(* Logix 5000 project; controller CTRL_PLC_V30 vendor 1 type 14 code 212 rev 34.11; software revision 34.02; part 2 of 2 *)
(* tags used below, declared in another part *)
   Aantal_RondjesT1 : DINT;
   Aantal_RondjesT2 : DINT;
   As_Test1_CTRL : AXIS_CIP_DRIVE;
   As_Test2_CTRL : AXIS_CIP_DRIVE;
   AsTest1Accel : REAL;
   AsTest1Snelheid : REAL;
   AsTest1StartPos : REAL;
   AsTest1StopPos : REAL;
   AsTest2Accel : REAL;
   AsTest2Snelheid : REAL;
   AsTest2StartPos : REAL;
   AsTest2StopPos : REAL;
   BOOL : BOOL;
   Drive_SAFE_OFF1 : ALIAS FOR DRIVER:SO.SafeTorqueOff1;
   Drive_SAFE_OFF2 : ALIAS FOR DRIVER:SO.SafeTorqueOff2;
   ERROR : BOOL;
   ERROR_1 : BOOL;
   ERROR_2 : BOOL;
   ESTP_ACTIVATED : BOOL;
   HomeT1 : ALIAS FOR IOP_HMI_BT[0].2;
   HomeT2 : ALIAS FOR IOP_HMI_BT[1].2;
   ILB_RESET_SAFETY1 : BOOL;
   ILG_CTRL_VOLT1 : BOOL;
   IO_SPLC_TO_CTRL : UDT_COMM_SPLC_TO_CTRL;
   IOP_HMI_BT : DINT[2];
   IOP_HMI_REAL : REAL[20];
   MDA_DATACHOICE : INT;
   MDB_DATACHOICE : INT;
   Motioncontrol13 : MOTION_INSTRUCTION;
   Motioncontrol14 : MOTION_INSTRUCTION;
   Motioncontrol21 : MOTION_INSTRUCTION;
   Motioncontrol26 : MOTION_INSTRUCTION;
   Motioncontrol27 : MOTION_INSTRUCTION;
   Motioncontrol3 : MOTION_INSTRUCTION;
   Motioncontrol30 : MOTION_INSTRUCTION;
   Motioncontrol4 : MOTION_INSTRUCTION;
   Motionctrl1 : MOTION_INSTRUCTION;
   Motionctrl2 : MOTION_INSTRUCTION;
   Motionstart1 : MOTION_INSTRUCTION;
   Motionstartl2 : MOTION_INSTRUCTION;
   OvertravelFault : BOOL;
   OvertravelFault2 : BOOL;
   QOP_HMI_BT : DINT[10];
   QOP_HMI_GRAPH1_HDR : REAL[10];
   QOP_HMI_GRAPH1_LINE1_DATAX : REAL[800];
   QOP_HMI_GRAPH1_LINE1_DATAY : REAL[800];
   QOP_HMI_GRAPH1_LINE1_HDR : REAL[10];
   QOP_HMI_GRAPH1_LINE2_DATAY : REAL[800];
   QOP_HMI_GRAPH2_HDR : REAL[10];
   QOP_HMI_GRAPH2_LINE1_DATAX : REAL[800];
   QOP_HMI_GRAPH2_LINE1_DATAY : REAL[800];
   QOP_HMI_GRAPH2_LINE2_DATAY : REAL[800];
   RondjesT1 : REAL;
   RondjesT2 : REAL;
   SAF_RESET_KNOP : BOOL;
   Safeovertravel1 : REAL;
   Safeovertravel2 : REAL;
   SAFETY_DOOR1_OPEN : BOOL;
   SAFETY_DOOR2_OPEN : BOOL;
   StartG : ALIAS FOR RIO_CTRL:3:I.0;
   StartLampje : ALIAS FOR RIO_CTRL:5:O.0;
   StartT1 : ALIAS FOR IOP_HMI_BT[0].0;
   StartT2 : ALIAS FOR IOP_HMI_BT[1].0;
   StateT1Routine : DINT;
   StateT2Routine : DINT;

   StopLampje : ALIAS FOR RIO_CTRL:5:O.1;
   StopR : ALIAS FOR RIO_CTRL:3:I.1;
   StopT1 : ALIAS FOR IOP_HMI_BT[0].1;
   StopT2 : ALIAS FOR IOP_HMI_BT[1].1;
   TEST_1x : BOOL;
   TIME_LATCH : BOOL; {access Read Only}
   Timer1 : TIMER := (PRE := 2);
   TIMER10 : TIMER := (PRE := 10000); {access Read Only}
   Timer2 : TIMER := (PRE := 2);
   Timeras1 : FBD_TIMER := (TimerEnable := 1, PRE := 9000, Reset := 1, ACC := 7821, EN := 1, TT := 1);
   Timeras2 : FBD_TIMER;
   Timeras3 : FBD_TIMER;
   Timeras4 : FBD_TIMER;
   Timeras5 : FBD_TIMER;
   Timeras6 : FBD_TIMER := (TimerEnable := 1, PRE := 200, Reset := 1, ACC := 151, EN := 1, TT := 1);
   Timeras7 : FBD_TIMER := (TimerEnable := 1, PRE := 9000, Reset := 1, ACC := 5957, EN := 1, TT := 1);
   Timeras8 : FBD_TIMER := (TimerEnable := 1, PRE := 9000, Reset := 1, ACC := 5010, EN := 1, TT := 1);
   Timeras9 : FBD_TIMER := (TimerEnable := 1, PRE := 9000, Reset := 1, ACC := 5001, EN := 1, TT := 1);
END_VAR

PROGRAM DataVersturen   (* main routine DataPLC *)
VAR
   FORLOOPINT : INT := 400; {access None}
   FORLOOPINT2 : DINT := 800; {access None}
   GRAPH1_LATESTX : INT; {access None}
   IDLE : DINT;
   POSITION1_INT : INT; {access None}
   POSITION2_INT : INT := 799; {access None}
   STEPSIZE2_LINE1 : REAL := -0.02; {access None}
   STEPSIZE_LINE1 : REAL := 11.875; {access None}
   TIMERMOV : TIMER := (PRE := 500, ACC := 10);
END_VAR

ROUTINE DataPLC   (* ladder *)
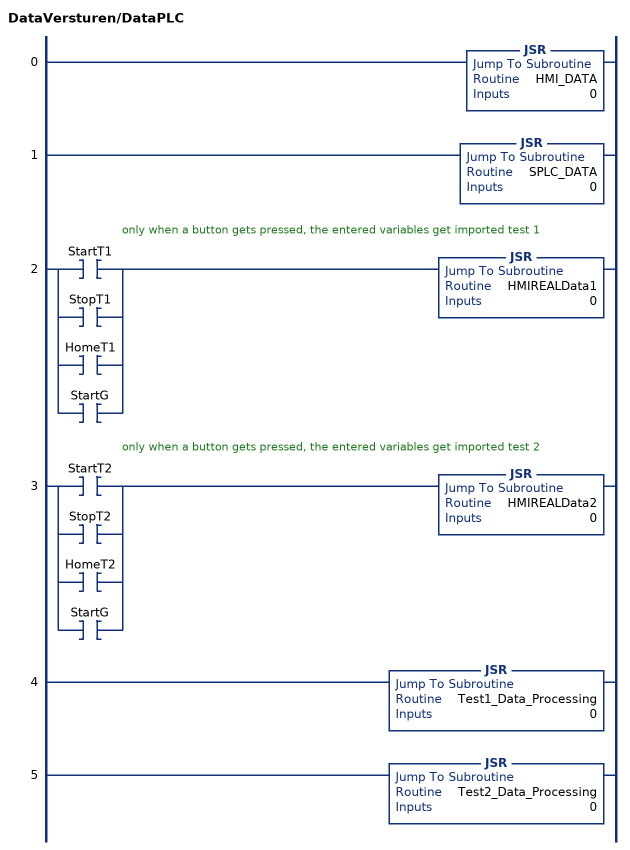
   0: JSR(HMI_DATA,0);
   1: JSR(SPLC_DATA,0);
   // only when a button gets pressed, the entered variables get imported test 1
   2: [XIC(StartT1) ,[XIC(StopT1) ,[XIC(HomeT1) ,XIC(StartG) ] ] ]JSR(HMIREALData1,0);
   // only when a button gets pressed, the entered variables get imported test 2
   3: [XIC(StartT2) ,[XIC(StopT2) ,[XIC(HomeT2) ,XIC(StartG) ] ] ]JSR(HMIREALData2,0);
   4: JSR(Test1_Data_Processing,0);
   5: JSR(Test2_Data_Processing,0);
END_ROUTINE

ROUTINE HMI_DATA   (* ladder *)
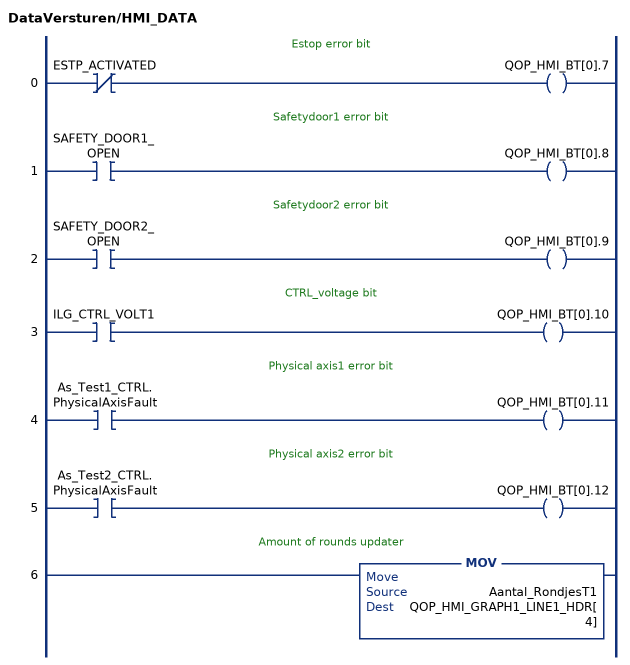
   // Estop error bit
   0: XIO(ESTP_ACTIVATED)OTE(QOP_HMI_BT[0].7);
   // Safetydoor1 error bit
   1: XIC(SAFETY_DOOR1_OPEN)OTE(QOP_HMI_BT[0].8);
   // Safetydoor2 error bit
   2: XIC(SAFETY_DOOR2_OPEN)OTE(QOP_HMI_BT[0].9);
   // CTRL_voltage bit
   3: XIC(ILG_CTRL_VOLT1)OTE(QOP_HMI_BT[0].10);
   // Physical axis1 error bit
   4: XIC(As_Test1_CTRL.PhysicalAxisFault)OTE(QOP_HMI_BT[0].11);
   // Physical axis2 error bit
   5: XIC(As_Test2_CTRL.PhysicalAxisFault)OTE(QOP_HMI_BT[0].12);
   // Amount of rounds updater
   6: MOV(Aantal_RondjesT1,QOP_HMI_GRAPH1_LINE1_HDR[4]);
END_ROUTINE

ROUTINE HMIREALData1   (* ladder *)
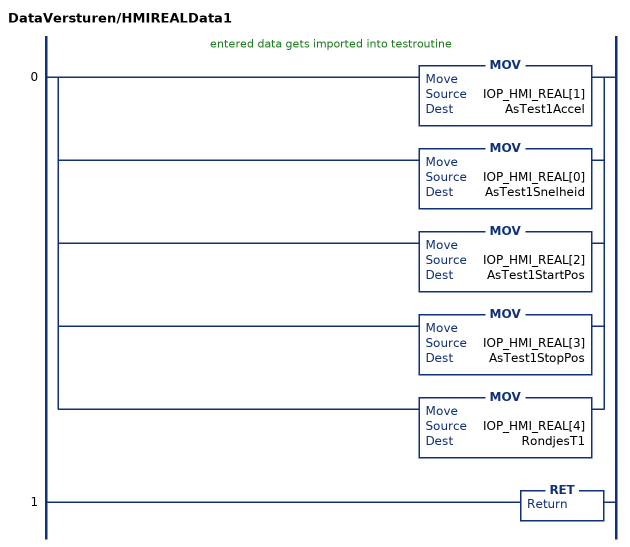
   // entered data gets imported into testroutine
   0: [MOV(IOP_HMI_REAL[1],AsTest1Accel) ,[MOV(IOP_HMI_REAL[0],AsTest1Snelheid) ,[MOV(IOP_HMI_REAL[2],AsTest1StartPos) ,[MOV(IOP_HMI_REAL[3],AsTest1StopPos) ,MOV(IOP_HMI_REAL[4],RondjesT1) ] ] ] ];
   1: RET();
END_ROUTINE

ROUTINE HMIREALData2   (* ladder *)
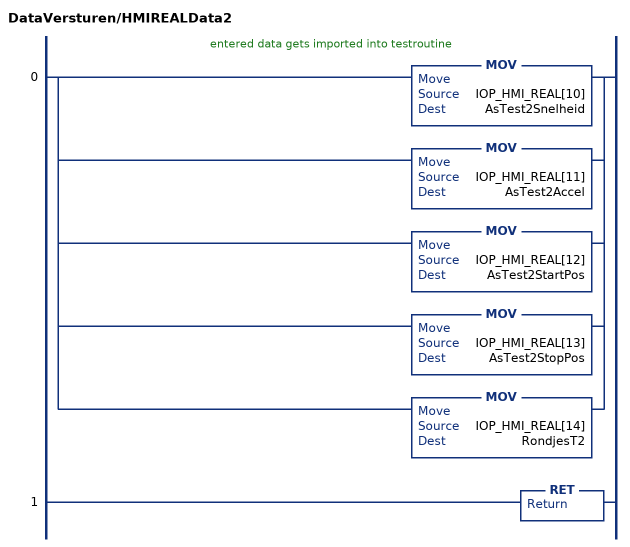
   // entered data gets imported into testroutine
   0: [MOV(IOP_HMI_REAL[10],AsTest2Snelheid) ,[MOV(IOP_HMI_REAL[11],AsTest2Accel) ,[MOV(IOP_HMI_REAL[12],AsTest2StartPos) ,[MOV(IOP_HMI_REAL[13],AsTest2StopPos) ,MOV(IOP_HMI_REAL[14],RondjesT2) ] ] ] ];
   1: RET();
END_ROUTINE

ROUTINE SPLC_DATA   (* ladder *)
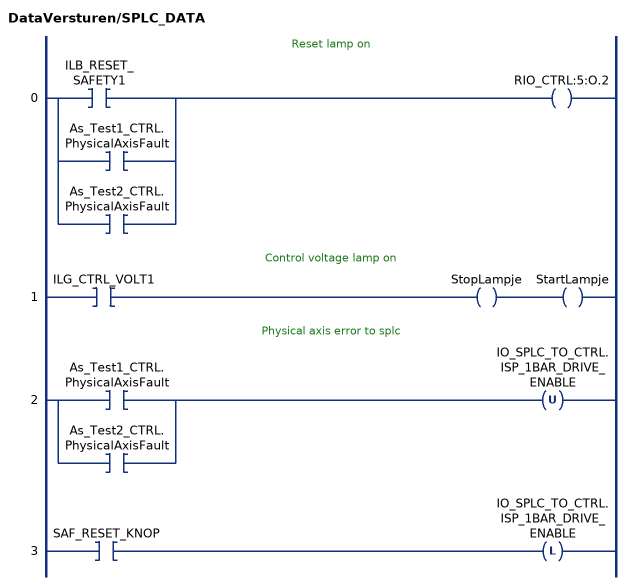
   // Reset lamp on
   0: [XIC(ILB_RESET_SAFETY1) ,[XIC(As_Test1_CTRL.PhysicalAxisFault) ,XIC(As_Test2_CTRL.PhysicalAxisFault) ] ]OTE(RIO_CTRL:5:O.2);
   // Control voltage lamp on
   1: XIC(ILG_CTRL_VOLT1)OTE(StopLampje)OTE(StartLampje);
   // Physical axis error to splc
   2: [XIC(As_Test1_CTRL.PhysicalAxisFault) ,XIC(As_Test2_CTRL.PhysicalAxisFault) ]OTU(IO_SPLC_TO_CTRL.ISP_1BAR_DRIVE_ENABLE);
   3: XIC(SAF_RESET_KNOP)OTL(IO_SPLC_TO_CTRL.ISP_1BAR_DRIVE_ENABLE);
END_ROUTINE

ROUTINE Test1_Data_Processing   (* structured text *)
   // wanneer state voltooid, dan naar volgende state
   
   CASE StateT1Routine OF
   	0: // idle state
   
   	1: // runs one time when subroutine starts
   	POSITION1_INT := 0;
   	FOR FORLOOPINT := 0 TO 799 BY 1 DO
   		QOP_HMI_GRAPH1_LINE1_DATAY[FORLOOPINT] := 0;		// emptying Array
   		QOP_HMI_GRAPH1_LINE2_DATAY[FORLOOPINT] := 0;		// emptying Array
   	END_FOR;
   	StateT1Routine := 2; // go to T1 state 2
   
   	2: // calculate steppsize
   	STEPSIZE_LINE1 := (AsTest1StopPos - AsTest1StartPos)/800;
   	STEPSIZE_LINE1 := STEPSIZE_LINE1 -0.0;
   	QOP_HMI_GRAPH1_LINE1_DATAX[0]:= AsTest1StartPos + 0.1;
   	FOR FORLOOPINT := 1 TO 799 BY 1 DO
   		QOP_HMI_GRAPH1_LINE1_DATAX[FORLOOPINT] := QOP_HMI_GRAPH1_LINE1_DATAX[FORLOOPINT-1]+STEPSIZE_LINE1;		// emtying Array
   	END_FOR;
   	QOP_HMI_GRAPH1_LINE1_DATAX[799]:= AsTest1StopPos - 0.1;
   	QOP_HMI_GRAPH1_HDR[2] := AsTest1StartPos;
   	QOP_HMI_GRAPH1_HDR[3]  :=AsTest1StopPos;
   	POSITION1_INT := 0;
   	StateT1Routine := 21;	// go to Test1Routine home sequence
   
   	6: // recording Data
   	StateT1Routine := 50 + MDA_DATACHOICE;
   
   	11:	// recording data
   	POSITION1_INT := 799;			//setting value ready for next state
   	StateT1Routine := 60 + MDA_DATACHOICE;
   
   	12: //changing graph setting
   	POSITION1_INT := 0;
   	QOP_HMI_GRAPH1_HDR[5] := 2;		// setting Ymax to a low value
   	FOR FORLOOPINT := 0 TO 399 BY 1 DO				// setting graph hight
   		IF QOP_HMI_GRAPH1_LINE1_DATAY[FORLOOPINT] > QOP_HMI_GRAPH1_HDR[5] THEN
   			QOP_HMI_GRAPH1_HDR[5] := QOP_HMI_GRAPH1_LINE1_DATAY[FORLOOPINT];
   		END_IF;
   	END_FOR;
   	FOR FORLOOPINT := 0 TO 399 BY 1 DO
   		IF QOP_HMI_GRAPH1_LINE2_DATAY[FORLOOPINT] > QOP_HMI_GRAPH1_HDR[5] THEN
   			QOP_HMI_GRAPH1_HDR[5] := QOP_HMI_GRAPH1_LINE2_DATAY[FORLOOPINT];
   		END_IF;
   	END_FOR;
   	IF (AsTest1StopPos - AsTest1StartPos)> 600 THEN // choosing graph x axis steppsize
   	QOP_HMI_GRAPH1_HDR[6]:= 20;
   	ELSIF (AsTest1StopPos - AsTest1StartPos)> 400 THEN
   	QOP_HMI_GRAPH1_HDR[6]:= 10;
   	ELSE
   	QOP_HMI_GRAPH1_HDR[6]:= 1;
   	END_IF;
   	IF QOP_HMI_GRAPH1_HDR[5] > 500 THEN				// choosing graph y axis steppsize
   	QOP_HMI_GRAPH1_HDR[7] := 50;
   	ELSIF QOP_HMI_GRAPH1_HDR[5] > 200 THEN
   	QOP_HMI_GRAPH1_HDR[7] := 25;
   	ELSIF QOP_HMI_GRAPH1_HDR[5] > 60 THEN
   	QOP_HMI_GRAPH1_HDR[7] := 5;
   	ELSE
   	QOP_HMI_GRAPH1_HDR[7] := 1;
   	END_IF;
   	StateT1Routine := 13; // go to Test1Routine state 13
   
   	14:	// check if all data has been sent to HMI
   	StateT1Routine := 15; // go to Test1Routine state 15
   
   	50:  // motion process
   	IF Motioncontrol3.PC THEN StateT1Routine := 10;	END_IF;
   
   	51: // Data of torque reference
   	IF As_Test1_CTRL.ActualPosition >= QOP_HMI_GRAPH1_LINE1_DATAX[POSITION1_INT] THEN
   		QOP_HMI_GRAPH1_LINE1_DATAY[POSITION1_INT]:= ABS(As_Test1_CTRL.TorqueReference);
   		POSITION1_INT := POSITION1_INT + 1;
   	END_IF;
   	IF POSITION1_INT > 799 OR Motioncontrol3.PC THEN
   		StateT1Routine := 10; // go to Test1Routine state 10
   	END_IF;
   
   	52: // Data of current reference
   	IF As_Test1_CTRL.ActualPosition >= QOP_HMI_GRAPH1_LINE1_DATAX[POSITION1_INT] THEN
   		QOP_HMI_GRAPH1_LINE1_DATAY[POSITION1_INT]:= ABS(As_Test1_CTRL.CurrentReference);
   		POSITION1_INT := POSITION1_INT + 1;
   
   	END_IF;
   	IF POSITION1_INT > 799 OR Motioncontrol3.PC THEN
   		StateT1Routine := 10; // go to Test1Routine state 10
   	END_IF;
   
   	53: // Data of actual velocity
   	IF As_Test1_CTRL.ActualPosition >= QOP_HMI_GRAPH1_LINE1_DATAX[POSITION1_INT] THEN
   		QOP_HMI_GRAPH1_LINE1_DATAY[POSITION1_INT]:= ABS(As_Test1_CTRL.ActualVelocity);
   		POSITION1_INT := POSITION1_INT + 1;
   
   	END_IF;
   	IF POSITION1_INT > 799 OR Motioncontrol3.PC THEN
   		StateT1Routine := 10; // go to Test1Routine state 10
   	END_IF;
   
   	60: // motion process
   	IF Motioncontrol4.PC THEN StateT1Routine := 12;	END_IF;
   
   	61: //TorqueReference
   	IF As_Test1_CTRL.ActualPosition <= QOP_HMI_GRAPH1_LINE1_DATAX[POSITION1_INT] THEN
   		QOP_HMI_GRAPH1_LINE2_DATAY[POSITION1_INT]:= ABS(As_Test1_CTRL.TorqueReference);
   		POSITION1_INT := POSITION1_INT - 1;
   	END_IF;
   	IF POSITION1_INT < 0 OR Motioncontrol4.PC THEN
   		StateT1Routine := 12; // go to T1 state 12
   	END_IF;
   
   	62: //CurrentReference
   	IF As_Test1_CTRL.ActualPosition <= QOP_HMI_GRAPH1_LINE1_DATAX[POSITION1_INT] THEN
   		QOP_HMI_GRAPH1_LINE2_DATAY[POSITION1_INT]:= ABS(As_Test1_CTRL.CurrentReference);
   		POSITION1_INT := POSITION1_INT - 1;
   	END_IF;
   	IF POSITION1_INT < 0 OR Motioncontrol4.PC THEN
   		StateT1Routine := 12; // go to T1 state 12
   	END_IF;
   
   	63: //ActualVelocity
   	IF As_Test1_CTRL.ActualPosition <= QOP_HMI_GRAPH1_LINE1_DATAX[POSITION1_INT] THEN
   		QOP_HMI_GRAPH1_LINE2_DATAY[POSITION1_INT]:= ABS(As_Test1_CTRL.ActualVelocity);
   		POSITION1_INT := POSITION1_INT - 1;
   	END_IF;
   	IF POSITION1_INT < 0 OR Motioncontrol4.PC THEN
   		StateT1Routine := 12; // go to T1 state 12
   	END_IF;
   
   END_CASE;
END_ROUTINE

ROUTINE Test2_Data_Processing   (* structured text *)
   // wanneer state voltooid, dan naar volgende state
   CASE StateT2Routine OF
   	0: // idle state
   
   	1: // runs one time when the subroutine starts
   	POSITION2_INT := 0;
   	FOR FORLOOPINT2 := 0 TO 799 BY 1 DO
   		QOP_HMI_GRAPH2_LINE1_DATAY[FORLOOPINT2] := 0;		// emtying Array
   		QOP_HMI_GRAPH2_LINE2_DATAY[FORLOOPINT2] := 0;		// emtying Array
   	END_FOR;
   	StateT2Routine := 2; // go to T2 state 2
   
   
   	2: // calculate steppsize
   	STEPSIZE2_LINE1 := (AsTest2StopPos - AsTest2StartPos)/800;
   	STEPSIZE2_LINE1 := STEPSIZE2_LINE1 -0.02;
   	QOP_HMI_GRAPH2_LINE1_DATAX[0]:= AsTest2StartPos + 0.1;
   	FOR FORLOOPINT2 := 1 TO 799 BY 1 DO
   		QOP_HMI_GRAPH2_LINE1_DATAX[FORLOOPINT2] := QOP_HMI_GRAPH2_LINE1_DATAX[FORLOOPINT2-1]+STEPSIZE2_LINE1;		// emtying Array
   	END_FOR;
   	QOP_HMI_GRAPH2_LINE1_DATAX[799]:= AsTest2StopPos - 0.1;
   	QOP_HMI_GRAPH2_HDR[2] := AsTest2StartPos;
   	QOP_HMI_GRAPH2_HDR[3]  :=AsTest2StopPos;
   	POSITION2_INT := 0;
   	StateT2Routine := 21; // go to Test2Routine state 20
   
   	6: // recording Data
   	StateT2Routine := 50 + MDB_DATACHOICE;
   
   	11:	// recording data
   	POSITION2_INT := 799;	//setting value ready for next state
   	StateT2Routine := 60 + MDB_DATACHOICE;
   
   	12: //changing graph setting
   	POSITION2_INT := 0;
   	QOP_HMI_GRAPH2_HDR[5] := 2;		// setting Ymax to a low value
   	FOR FORLOOPINT2 := 0 TO 799 BY 1 DO				// setting graph hight
   		IF QOP_HMI_GRAPH2_LINE1_DATAY[FORLOOPINT2] > QOP_HMI_GRAPH2_HDR[5] THEN
   			QOP_HMI_GRAPH2_HDR[5] := QOP_HMI_GRAPH2_LINE1_DATAY[FORLOOPINT2];
   		END_IF;
   	END_FOR;
   	FOR FORLOOPINT2 := 0 TO 799 BY 1 DO
   		IF QOP_HMI_GRAPH2_LINE2_DATAY[FORLOOPINT2] > QOP_HMI_GRAPH2_HDR[5] THEN
   			QOP_HMI_GRAPH2_HDR[5] := QOP_HMI_GRAPH2_LINE2_DATAY[FORLOOPINT2];
   		END_IF;
   	END_FOR;
   	IF (AsTest2StopPos - AsTest2StartPos)> 600 THEN // choosing graph x axis steppsize
   	QOP_HMI_GRAPH2_HDR[6]:= 20;
   	ELSIF (AsTest2StopPos - AsTest2StartPos)> 400 THEN
   	QOP_HMI_GRAPH2_HDR[6]:= 10;
   	ELSE
   	QOP_HMI_GRAPH2_HDR[6]:= 1;
   	END_IF;
   	IF QOP_HMI_GRAPH2_HDR[5] > 500 THEN				// choosing graph y axis steppsize
   	QOP_HMI_GRAPH2_HDR[7] := 50;
   	ELSIF QOP_HMI_GRAPH2_HDR[5] > 200 THEN
   	QOP_HMI_GRAPH2_HDR[7] := 25;
   	ELSIF QOP_HMI_GRAPH2_HDR[5] > 60 THEN
   	QOP_HMI_GRAPH2_HDR[7] := 5;
   	ELSE
   	QOP_HMI_GRAPH2_HDR[7] := 1;
   	END_IF;
   	StateT2Routine := 13; // go to Test2Routine state 13
   
   	14:	// check if all data has been sent to HMI
   	StateT2Routine := 15; // go to Test2Routine state 15
   
   	50:
   	IF Motioncontrol13.PC THEN StateT2Routine := 10;	END_IF;
   
   	51: //TorqueReference
   	IF As_Test2_CTRL.ActualPosition >= QOP_HMI_GRAPH2_LINE1_DATAX[POSITION2_INT] THEN
   		QOP_HMI_GRAPH2_LINE1_DATAY[POSITION2_INT]:= ABS(As_Test2_CTRL.TorqueReference);
   		POSITION2_INT := POSITION2_INT + 1;
   	END_IF;
   	IF POSITION2_INT > 799 OR Motioncontrol13.PC THEN
   		StateT2Routine := 10; // go to Test2Routine state 10
   	END_IF;
   
   	52: //CurrentReference
   	IF As_Test2_CTRL.ActualPosition >= QOP_HMI_GRAPH2_LINE1_DATAX[POSITION2_INT] THEN
   		QOP_HMI_GRAPH2_LINE1_DATAY[POSITION2_INT]:= ABS(As_Test2_CTRL.CurrentReference);
   		POSITION2_INT := POSITION2_INT + 1;
   	END_IF;
   	IF POSITION2_INT > 799 OR Motioncontrol13.PC THEN
   		StateT2Routine := 10; // go to Test2Routine state 10
   	END_IF;
   	53: //ActualVelocity
   	IF As_Test2_CTRL.ActualPosition >= QOP_HMI_GRAPH2_LINE1_DATAX[POSITION2_INT] THEN
   		QOP_HMI_GRAPH2_LINE1_DATAY[POSITION2_INT]:= ABS(As_Test2_CTRL.ActualVelocity);
   		POSITION2_INT := POSITION2_INT + 1;
   	END_IF;
   	IF POSITION2_INT > 799 OR Motioncontrol13.PC THEN
   		StateT2Routine := 10; // go to Test2Routine state 10
   	END_IF;
   
   	60: // motion sequence
   	IF Motioncontrol14.PC THEN StateT2Routine := 12;
   	END_IF;
   
   	61: //TorqueReference
   	IF As_Test2_CTRL.ActualPosition <= QOP_HMI_GRAPH2_LINE1_DATAX[POSITION2_INT] THEN
   		QOP_HMI_GRAPH2_LINE2_DATAY[POSITION2_INT]:= ABS(As_Test2_CTRL.TorqueReference);
   		POSITION2_INT := POSITION2_INT - 1;
   	END_IF;
   	IF POSITION2_INT < 0 OR Motioncontrol14.PC THEN
   		StateT2Routine := 12; // go to T2 state 12
   	END_IF;
   
   	62: //CurrentReference
   	IF As_Test2_CTRL.ActualPosition <= QOP_HMI_GRAPH2_LINE1_DATAX[POSITION2_INT] THEN
   		QOP_HMI_GRAPH2_LINE2_DATAY[POSITION2_INT]:= ABS(As_Test2_CTRL.CurrentReference);
   		POSITION2_INT := POSITION2_INT - 1;
   	END_IF;
   	IF POSITION2_INT < 0 OR Motioncontrol14.PC THEN
   		StateT2Routine := 12; // go to T2 state 12
   	END_IF;
   
   	63: //ActualVelocity
   	IF As_Test2_CTRL.ActualPosition <= QOP_HMI_GRAPH2_LINE1_DATAX[POSITION2_INT] THEN
   		QOP_HMI_GRAPH2_LINE2_DATAY[POSITION2_INT]:= ABS(As_Test2_CTRL.ActualVelocity);
   		POSITION2_INT := POSITION2_INT - 1;
   	END_IF;
   	IF POSITION2_INT < 0 OR Motioncontrol14.PC THEN
   		StateT2Routine := 12; // go to T2 state 12
   	END_IF;
   END_CASE;
END_ROUTINE
END_PROGRAM

PROGRAM MainProgram   (* main routine MainRoutine *)
VAR
   Axis1AtHome : ALIAS FOR As_Test1_CTRL.HomingStatus;
   Axis2AtHome : ALIAS FOR As_Test2_CTRL.HomingStatus;
   FORLOOPINT : INT := 1000; {access None}
   Motioncontrol1 : MOTION_INSTRUCTION := (FLAGS := -1476395008, EN := 1, DN := 1, PC := 1);
   Motioncontrol2 : MOTION_INSTRUCTION := (FLAGS := -1610612736, EN := 1, DN := 1, STATE := 1);
   StateHome1 : DINT;
   StateHome2 : DINT;
   StateMain : DINT := 8;
   Test1_Snelheid_HMI : DINT;
   Test2_Snelheid_HMI : DINT;
END_VAR

ROUTINE AsFout1   (* structured text *)
   IF SAF_RESET_KNOP THEN // if ctrl voltage is on, request reset
   	MAFR(As_Test1_CTRL,Motioncontrol1);
   	OvertravelFault := 0;
   END_IF;
   
END_ROUTINE

ROUTINE AsFout2   (* structured text *)
   IF SAF_RESET_KNOP THEN // if ctrl voltage is on, request reset
   	MAFR(As_Test2_CTRL,Motioncontrol2);
   	OvertravelFault2 := 0;
   END_IF;
   
END_ROUTINE

ROUTINE AxisHoming1   (* structured text *)
   CASE StateHome1 OF
   
   	0: //idle state
   
   	1: MAH(As_Test1_CTRL,Motioncontrol21); // start homesequence
   		Safeovertravel1 := As_Test1_CTRL.ActualPosition;
   		StateHome1 := 2; // go to home1 state 2
   
   	2: IF Motioncontrol21.PC AND As_Test1_CTRL.AxisHomedStatus THEN // handshake for making sure the axis is really at home
   			StateHome1 := 0; // go to home1 idle state
   		ELSIF As_Test1_CTRL.ActualPosition <= (Safeovertravel1 - 2000) then
   			MAS(As_Test1_CTRL,Motioncontrol1,0,no,1000,Unitspersec2,no,1000,Unitspersec3);
   			OvertravelFault := 1;
   			StateHome1 := 0; // go to home1 idle state
   		END_IF;
   END_CASE;
   
   
   
   
   
   
   
END_ROUTINE

ROUTINE AxisHoming2   (* structured text *)
   CASE StateHome2 OF
   
   	0: 	//Idle state
   
   	1: MAH(As_Test2_CTRL,Motioncontrol30); // start homesequence
   		Safeovertravel2 := As_Test2_CTRL.ActualPosition;
   		StateHome2 := 2; // go to home2 state 2
   
   	2: IF Motioncontrol30.PC AND As_Test2_CTRL.AxisHomedStatus THEN // handshake for making sure the axis is really at home
   		StateHome2 := 0; // go to home2 idle state
   		ELSIF As_Test2_CTRL.ActualPosition <= (Safeovertravel2 - 2000) then
   		 	MAS(As_Test2_CTRL,Motioncontrol2,0,no,1000,Unitspersec2,no,1000,Unitspersec3);
   			OvertravelFault2 := 1;
   			StateHome2 := 0; // go to home2 idle state
   		END_IF;
   END_CASE;
   
   
   
   
   
   
   
END_ROUTINE

ROUTINE MainRoutine   (* structured text *)
   // when state, next state
   CASE StateMain OF
   
   	0: StateT1Routine := 0;   // Error state
   		StateT2Routine := 0;
   		StateHome1 := 0;
   		StateHome2 := 0;
   
   
   		Timeras6.Reset := 0;  // timer to prevent error routine overload
   		TONR(Timeras6);
   		Timeras6.PRE:= 200;
   		IF NOT Timeras6.DN THEN
   			Timeras6.TimerEnable := 1;
   		ELSE
   			Timeras6.TimerEnable := 0;
   		END_IF;
   
   		IF Timeras6.ACC >150 THEN
   			IF (As_Test1_CTRL.PhysicalAxisFault OR As_Test1_CTRL.MotionFault)  AND ILG_CTRL_VOLT1 THEN // check error axis 1
   				StateMain := 8;
   			elsif (As_Test2_CTRL.PhysicalAxisFault OR As_Test2_CTRL.MotionFault) AND ILG_CTRL_VOLT1 then // check error axis 2
   				StateMain := 9;
   			ELSIF ILG_CTRL_VOLT1 THEN // check control voltage, servomotor on
   				MSO(As_Test1_CTRL, Motionctrl1 );
   				MSO(As_Test2_CTRL, Motionctrl2 );
   				StateMain := 1; // go to main idle state
   			END_IF;
   			Timeras6.Reset := 1;
   		end_if;
   
   		StateT1Routine := 0; // back to standard values
   		StateT2Routine := 0;
   		StateHome1 := 0;
   		StateHome2 := 0;
   
   	1: MSO(As_Test1_CTRL, Motionstart1 );  // State 1 idle state, motor on to prevent errors
   		MSO(As_Test2_CTRL, Motionstartl2 );
   		IF StartT1 THEN  // when button test 1 go to testroutine1
   			StateMain := 2; // go to stateMain 2
   		ELSIF StartT2 THEN  // when button test 2 go to testroutine2
   			StateMain := 3; // go to stateMain 3
   		ELSIF HomeT1 THEN // when button home1 go to homeroutine1
   			StateMain := 4; // go to stateMain 4
   		ELSIF HomeT2 THEN // when button home 2 go to homeroutine2
   			StateMain := 5;	// go to stateMain 5
   		ELSIF StopT1 THEN // when button stop1 go to stoproutine1
   			StateMain := 6; // go to stateMain 6
   		ELSIF StopT2 THEN // when button stop2 go to stoproutine2
   			StateMain := 7;	// go to stateMain 7
   		ELSIF (As_Test1_CTRL.PhysicalAxisFault OR As_Test1_CTRL.MotionFault) THEN 	 // when error axis 1 go to errorroutine1
   			StateMain := 8; // go to stateMain 8
   		ELSIF (As_Test2_CTRL.PhysicalAxisFault OR As_Test2_CTRL.MotionFault) THEN // when error axis 2 go to errorroutine2
   			StateMain := 9; // go to stateMain 9
   		ELSIF StopR THEN //stop both rails
   			StateMain := 10; //go to state main 10
   		ELSIF StartG THEN // start both motors
   			StateMain := 11; // go to state main 11
   		ELSIF NOT As_Test1_CTRL.Registration1InputStatus OR NOT As_Test1_CTRL.Registration2InputStatus THEN
   			JSR (StopAxis1);
   		ELSIF NOT As_Test2_CTRL.Registration1InputStatus OR NOT As_Test2_CTRL.Registration2InputStatus THEN
   			JSR (StopAxis2);
   		END_IF;
   
   		// keep calling rubroutines otherwise statediagram wont get finished
   		JSR(Test1Routine);
   		JSR(Test2Routine);
   		JSR(AxisHoming1);
   		JSR(AxisHoming2);
   
   	2:
   	StateT1Routine := 1; // from subroutine idle state to start test
   	Aantal_RondjesT1 := 0; // standard value
   	StateMain:= 1; // back to mainroutine idle state
   
   	3:
   	StateT2Routine := 1; // from subroutine idle state to start test
   	Aantal_RondjesT2 := 0; // standard value
   	StateMain:= 1; // back to mainroutine idle state
   
   	4:
   	StateHome1 := 1; // from subroutine idle state to homesequence
   	StateMain := 1; // back to mainroutine idle state
   
   	5:
   	StateHome2 := 1; // from subroutine idle state to homesequence
   	StateMain := 1; // back to mainroutine idle state
   
       6:
   	JSR(StopAxis1);
   	StateMain := 1; // back to mainroutine error state
   
   	7: // jump to subroutine StopAxis 2
   	JSR(StopAxis2);
   	StateMain := 1; // go to main state 1
   
   	8:
   	IF StopT1 THEN  // Making sure when in a state, stoproutine can always be called
   		JSR(StopAxis1);
   	ELSIF StopT2 THEN
   		JSR(StopAxis2);
   	END_IF;
   
   	Timeras1.Reset := 0; // timer because of the control voltage, this way the drive gets power and then after 5 sec resets
   	TONR(Timeras1);
   	Timeras1.PRE:= 9000;
   	IF NOT Timeras1.DN THEN
   		Timeras1.TimerEnable := 1;
   	ELSE
   		Timeras1.TimerEnable := 0;
   	END_IF;
   	IF Timeras1.ACC >5000 THEN
   	Timeras1.Reset := 1;
   	JSR(AsFout1);
   	END_IF;
   
   	IF NOT (As_Test1_CTRL.PhysicalAxisFault OR As_Test1_CTRL.MotionFault) THEN // handshake way where the drive gives a sign its ready
   		StateMain := 0; // go to main error state
   	end_if;
   
   
   	9:
   	IF StopT2 THEN // Making sure when in a state, stoproutine can always be called
   		JSR(StopAxis1);
   	ELSIF StopT2 THEN
   		JSR(StopAxis2);
   	END_IF;
   
   	Timeras8.Reset := 0; // timer because of the control voltage, this way the drive gets power and then after 5 sec resets
   	TONR(Timeras8);
   	Timeras8.PRE:= 9000;
   	IF NOT Timeras8.DN THEN
   		Timeras8.TimerEnable := 1;
   	ELSE
   		Timeras8.TimerEnable :=0;
   	END_IF;
   	IF Timeras8.ACC >5000 THEN
   	Timeras8.Reset := 1;
   	JSR(AsFout2);
   	END_IF;
   
   	IF NOT (As_Test2_CTRL.PhysicalAxisFault OR As_Test2_CTRL.MotionFault) THEN // handshake way where the drive gives a sign its ready
   		StateMain := 0;
   	end_if;
   
   	10:
   	IF StopR THEN  // Making sure when in a state, stoproutine can always be called
   		JSR(StopPhysical_1);
   	END_IF;
   
   	Timeras1.Reset := 0; // timer because of the control voltage, this way the drive gets power and then after 5 sec resets
   	TONR(Timeras1);
   	Timeras1.PRE:= 9000;
   	IF NOT Timeras1.DN THEN
   		Timeras1.TimerEnable := 1;
   	ELSE
   		Timeras1.TimerEnable := 0;
   	END_IF;
   	IF Timeras1.ACC >5000 THEN
   	Timeras1.Reset := 1;
   	JSR(AsFout1);
   	END_IF;
   
   	IF NOT (As_Test1_CTRL.PhysicalAxisFault OR As_Test1_CTRL.MotionFault) THEN // handshake way where the drive gives a sign its ready
   		StateMain := 0; // go to main error state
   	ELSIF
   	NOT (As_Test2_CTRL.PhysicalAxisFault OR As_Test2_CTRL.MotionFault) THEN // handshake way where the drive gives a sign its ready
   		StateMain := 0;
   	END_IF;
   
   	11: //start knop start allebei de opstellingen
   	StateT1Routine := 1;
   	Aantal_RondjesT1 := 0;
   	StateT2Routine := 1;
   	Aantal_RondjesT2 := 0;
   	StateMain:= 1;
   
   END_CASE;
END_ROUTINE

ROUTINE StopAxis1   (* structured text *)
   MAS(As_Test1_CTRL,Motioncontrol1,0,1,2000,Unitspersec2,0,2000,Unitspersec3); // axisstop command
   
   IF Motioncontrol1.PC AND As_Test1_CTRL.VelocityStandstillStatus THEN // making sure the servo is standing still, then turn off
   	//MSF(As_Test1_CTRL, Motioncontrol1 );
   	StateT1Routine := 0; // go to Test1Routine idle state
   END_IF;
   
END_ROUTINE

ROUTINE StopAxis2   (* structured text *)
   MAS(As_Test2_CTRL,Motioncontrol2,0,1,2000,Unitspersec2,no,2000,Unitspersec3); // stop command
   
   IF Motioncontrol2.PC AND As_Test2_CTRL.VelocityStandstillStatus THEN // making sure the servo is standing still, then turn off
   //	MSF(As_Test2_CTRL, Motioncontrol2 );
   	StateT2Routine := 0; // go to Test2Routine idle state
   END_IF;
   
END_ROUTINE

ROUTINE StopPhysical_1   (* structured text *)
   MAS(As_Test1_CTRL,Motioncontrol1,0,1,2000,Unitspersec2,0,2000,Unitspersec3); // axisstop command
   MAS(As_Test2_CTRL,Motioncontrol2,0,1,2000,Unitspersec2,0,2000,Unitspersec3); // axisstop command
   
   IF Motioncontrol1.PC AND As_Test1_CTRL.VelocityStandstillStatus THEN // making sure the servo is standing still, then turn off
   	//MSF(As_Test1_CTRL, Motioncontrol1 );
   	StateT1Routine := 0; // go to Test1Routine idle state
   ELSIF
   	Motioncontrol2.PC AND As_Test2_CTRL.VelocityStandstillStatus THEN // making sure the servo is standing still, then turn off
   	//MSF(As_Test1_CTRL, Motioncontrol1 );
   	StateT2Routine := 0; // go to Test1Routine idle state
   END_IF;
END_ROUTINE

ROUTINE Test1Routine   (* structured text *)
   // wanneer state voltooid, dan naar volgende state
   CASE StateT1Routine OF
   	0: // idle state
   
   	3: //Run To Start Position
   	MAM(As_Test1_CTRL,Motioncontrol4,0,AsTest1StartPos,1000,Unitspersec,1000,Unitspersec2,2000,Unitspersec2,SCurve,5000,5000,Unitspersec3,Disabled,Programmed,0,None,0,0); //HMI positie en HMI snelheid in negatieve directie
   	StateT1Routine := 4; // go to T1 state 4
   
   	4: // motion instruction
   	IF Motioncontrol4.PC THEN
   		StateT1Routine := 5; // go to T1 state 5
   	END_IF;
   
   	5: // Starting test, to end position
   	MAM(As_Test1_CTRL,Motioncontrol3,0,AsTest1StopPos,AsTest1Snelheid,Unitspersec,AsTest1Accel,Unitspersec2,AsTest1Accel,Unitspersec2,SCurve,5000,5000,Unitspersec3,Disabled,Programmed,0,None,0,0);
   	StateT1Routine := 6; // go to Test1_Data_Processing state 6
   
   	10: // back to start position
   	MAM(As_Test1_CTRL,Motioncontrol4,0,AsTest1StartPos,AsTest1Snelheid,Unitspersec,AsTest1Accel,Unitspersec2,AsTest1Accel,Unitspersec2,SCurve,5000,5000,Unitspersec3,Disabled,Programmed,0,None,0,0);
   	StateT1Routine := 11; // go to Test1_Data_Processing state 11
   
   	13: // amount of rounds done, every round plus one
   	Aantal_RondjesT1 := Aantal_RondjesT1 +1;
   	StateT1Routine := 14; // go to Test1_Data_Processing state 14
   
   	15: // compare if the amount of rounds is as much as configured
   	IF Motioncontrol4.PC  THEN
   		IF RondjesT1 <= Aantal_RondjesT1 THEN
   			StateT1Routine := 0;				// Back to T1 idle state
   		ELSE
   			StateT1Routine := 5;				// Start next Run
   		END_IF;
   	END_IF;
   
   	21: // motion instruction
   	IF Motioncontrol26.PC AND As_Test1_CTRL.VelocityStandstillStatus THEN
   		StateT1Routine := 3; // go to T1 state 3
   	ELSIF As_Test1_CTRL.ActualPosition <= (Safeovertravel1 - 1000) then
   	MAS(As_Test1_CTRL,Motioncontrol1,0,no,1000,Unitspersec2,no,1000,Unitspersec3);
   	OvertravelFault := 1;
   	StateT1Routine := 0; // go to T1 idle state
   	END_IF;
   END_CASE;
END_ROUTINE

ROUTINE Test2Routine   (* structured text *)
   // wanneer state voltooid, dan naar volgende state
   CASE StateT2Routine OF
   	0: // idle state
   
   	3: //Run To Start Position
   	MAM(As_Test2_CTRL,Motioncontrol14,0,AsTest2StartPos,1000,Unitspersec,1000,Unitspersec2,2000,Unitspersec2,SCurve,5000,5000,Unitspersec3,Disabled,Programmed,0,None,0,0); //HMI positie en HMI snelheid in negatieve directie
   	StateT2Routine := 4; // go to T2 state 4
   
   	4: // motion instruction
   	IF Motioncontrol14.PC THEN
   		StateT2Routine := 5; // go to T2 state 5
   	END_IF;
   
   	5:// Starting test, to end position
   	MAM(As_Test2_CTRL,Motioncontrol13,0,AsTest2StopPos,AsTest2Snelheid,Unitspersec,AsTest2Accel,Unitspersec2,AsTest2Accel,Unitspersec2,SCurve,5000,5000,Unitspersec3,Disabled,Programmed,0,None,0,0); //HMI positie en HMI snelheid in positieve directie
   	StateT2Routine := 6; // go to Test2_Data_Processing state 6
   
   	10: // back to start position
   	MAM(As_Test2_CTRL,Motioncontrol14,0,AsTest2StartPos,AsTest2Snelheid,Unitspersec,AsTest2Accel,Unitspersec2,AsTest2Accel,Unitspersec2,SCurve,5000,5000,Unitspersec3,Disabled,Programmed,0,None,0,0); //HMI positie en HMI snelheid in negatieve directie
   	StateT2Routine := 11; // go to Test2_Data_Processing state 11
   
   	13: // amount of rounds done, every round plus one
   	Aantal_RondjesT2 := Aantal_RondjesT2 +1;
   	StateT2Routine := 14; // go to Test2_Data_Processing state 14
   
   	15: // compare if the amount of rounds is as much as configured
   	IF Motioncontrol14.PC  THEN
   		IF RondjesT2 <= Aantal_RondjesT2 THEN
   			StateT2Routine := 0;				// Back to Test2 idle state
   		ELSE
   			StateT2Routine := 5;				// Start next Run
   		END_IF;
   	END_IF;
   
   	21: // motion instruction
   	IF Motioncontrol27.PC AND As_Test2_CTRL.VelocityStandstillStatus THEN
   		StateT2Routine := 3; // go to T2 state 3
   	ELSIF As_Test2_CTRL.ActualPosition <= (Safeovertravel2 - 1000) then
   		MAS(As_Test2_CTRL,Motioncontrol2,0,no,1000,Unitspersec2,no,1000,Unitspersec3);
   		OvertravelFault2 := 1;
   		StateT2Routine := 0; // go to T2 idle state
   	END_IF;
   END_CASE;
END_ROUTINE
END_PROGRAM

PROGRAM SafetyProgram   (* main routine MainRoutine, safety *)
VAR
   BUS_CTRL_VOLT_ON : ALIAS FOR RIO_CTRL:2:O.Pt02Data;
   CTRL_Volt_ON : ALIAS FOR RIO_CTRL:1:I.Pt04Data;
   Drive1EnableSignal : ALIAS FOR RIO_CTRL:2:O.Pt00Data;
   Drive2EnableSignal : ALIAS FOR RIO_CTRL:2:O.Pt01Data;
   DRIVE_SAF_ENABLE : BOOL;
   DRIVE_SAF_OFF_FEEDBACK2 : ALIAS FOR DRIVER:SI.TorqueDisabled2;
   DRIVE_SAFE_OFF_FEEDBACK1 : ALIAS FOR DRIVER:SI.TorqueDisabled1;
   DriveRESET1 : ALIAS FOR DRIVER:SO.Reset1;
   DriveRESET2 : ALIAS FOR DRIVER:SO.Reset2;
   Estp_Testkast : EMERGENCY_STOP := (ResetType := 1, ChannelA := 1, ChannelB := 1, O1 := 1);
   IPB_SAF_RESET_KNOP : ALIAS FOR RIO_CTRL:1:I.Pt05Data;
   SAF_Drive_SAFE_OFF : TIMER := (PRE := 800, ACC := 800, EN := 1, DN := 1);
   SAF_DRIVEDELAY_SAF_OK : BOOL := 1;
   SAF_DRIVESAF_OFF : BOOL;
   SAF_DRIVESAF_OK : BOOL;
   SAF_ESTP_1 : ALIAS FOR RIO_CTRL:1:I.Pt00Data;
   SAF_ESTP_2 : ALIAS FOR RIO_CTRL:1:I.Pt01Data;
   SAF_FAULT_RESET : BOOL;
   SAF_HMI_FAULT_RESET : BOOL;
   SAF_RESET_ESTOP : BOOL;
   SafetySchermA0 : ALIAS FOR RIO_CTRL:1:I.Pt02Data;
   SafetySchermA1 : ALIAS FOR RIO_CTRL:1:I.Pt03Data;
   SafetySchermB0 : ALIAS FOR RIO_CTRL:1:I.Pt06Data;
   SafetySchermB1 : ALIAS FOR RIO_CTRL:1:I.Pt07Data;
   SPLC_CTRL_VOLT_ON : BOOL;
   SPLC_DCS_DRIVE1 : DCI_STOP := (ChannelA := 1, ChannelB := 1, InputStatus := 1, ColdStartType := 1, SafetyFunction := 1, DiscrepancyTime := 200, O1 := 1);
   SPLC_DCS_DRIVE2 : DCI_STOP := (ChannelA := 1, ChannelB := 1, InputStatus := 1, ColdStartType := 1, SafetyFunction := 1, DiscrepancyTime := 200, O1 := 1);
   SPLC_ONS : BOOL;
   SPLC_ROUT_DRIVE_SAFEOFF1 : REDUNDANT_OUTPUT := (Enable := 1, O1FF := 1, O2FF := 1, FP := 1);
   SPLC_ROUT_DRIVE_SAFEOFF2 : REDUNDANT_OUTPUT := (Enable := 1, O1FF := 1, O2FF := 1, FP := 1);
END_VAR

ROUTINE CLR_FAULT   (* ladder *)
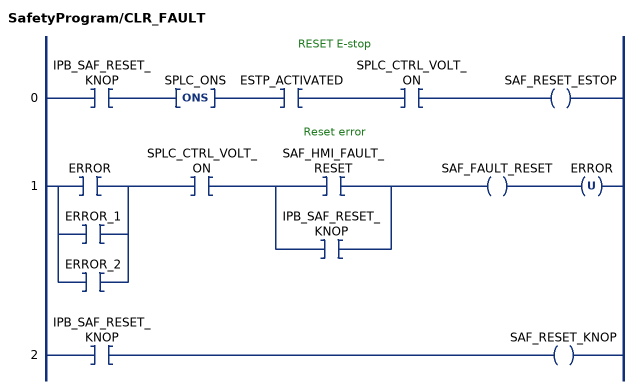
   // RESET E-stop
   0: XIC(IPB_SAF_RESET_KNOP)ONS(SPLC_ONS)XIC(ESTP_ACTIVATED)XIC(SPLC_CTRL_VOLT_ON)OTE(SAF_RESET_ESTOP);
   // Reset error
   1: [XIC(ERROR) ,[XIC(ERROR_1) ,XIC(ERROR_2) ] ]XIC(SPLC_CTRL_VOLT_ON)[XIC(SAF_HMI_FAULT_RESET) ,XIC(IPB_SAF_RESET_KNOP) ]OTE(SAF_FAULT_RESET)OTU(ERROR);
   2: XIC(IPB_SAF_RESET_KNOP)OTE(SAF_RESET_KNOP);
END_ROUTINE

ROUTINE CTRL_Voltage   (* ladder *)
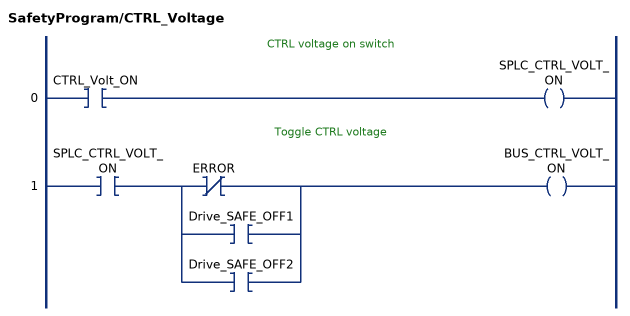
   // CTRL voltage on switch
   0: XIC(CTRL_Volt_ON)OTE(SPLC_CTRL_VOLT_ON);
   // Toggle CTRL voltage
   1: XIC(SPLC_CTRL_VOLT_ON)[XIO(ERROR) ,XIC(Drive_SAFE_OFF1) ,XIC(Drive_SAFE_OFF2) ]OTE(BUS_CTRL_VOLT_ON);
END_ROUTINE

ROUTINE Indicatielampjes   (* ladder *)
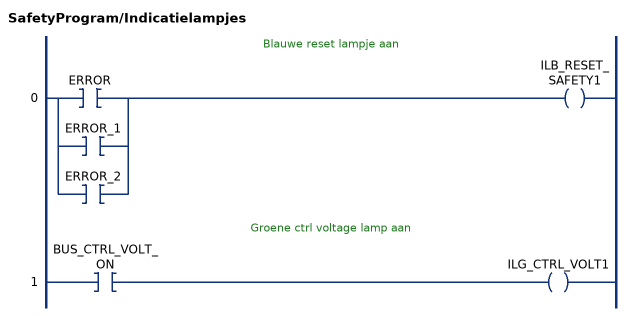
   // Blauwe reset lampje aan
   0: [XIC(ERROR) ,[XIC(ERROR_1) ,XIC(ERROR_2) ] ]OTE(ILB_RESET_SAFETY1);
   // Groene ctrl voltage lamp aan
   1: XIC(BUS_CTRL_VOLT_ON)OTE(ILG_CTRL_VOLT1);
END_ROUTINE

ROUTINE Kinetix_Drive_1   (* ladder *)
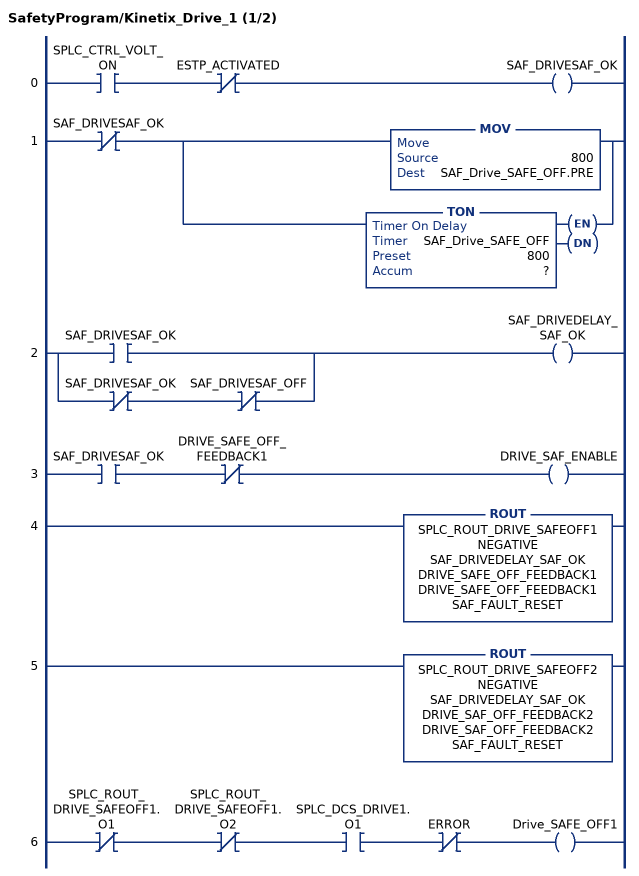
   0: XIC(SPLC_CTRL_VOLT_ON)XIO(ESTP_ACTIVATED)OTE(SAF_DRIVESAF_OK);
   1: XIO(SAF_DRIVESAF_OK)[MOV(800,SAF_Drive_SAFE_OFF.PRE) ,TON(SAF_Drive_SAFE_OFF,?,?) ];
   2: [XIC(SAF_DRIVESAF_OK) ,XIO(SAF_DRIVESAF_OK) XIO(SAF_DRIVESAF_OFF) ]OTE(SAF_DRIVEDELAY_SAF_OK);
   3: XIC(SAF_DRIVESAF_OK)XIO(DRIVE_SAFE_OFF_FEEDBACK1)OTE(DRIVE_SAF_ENABLE);
   4: ROUT(SPLC_ROUT_DRIVE_SAFEOFF1,NEGATIVE,SAF_DRIVEDELAY_SAF_OK,DRIVE_SAFE_OFF_FEEDBACK1,DRIVE_SAFE_OFF_FEEDBACK1,SAF_FAULT_RESET);
   5: ROUT(SPLC_ROUT_DRIVE_SAFEOFF2,NEGATIVE,SAF_DRIVEDELAY_SAF_OK,DRIVE_SAF_OFF_FEEDBACK2,DRIVE_SAF_OFF_FEEDBACK2,SAF_FAULT_RESET);
   6: XIO(SPLC_ROUT_DRIVE_SAFEOFF1.O1)XIO(SPLC_ROUT_DRIVE_SAFEOFF1.O2)XIC(SPLC_DCS_DRIVE1.O1)XIO(ERROR)OTE(Drive_SAFE_OFF1);
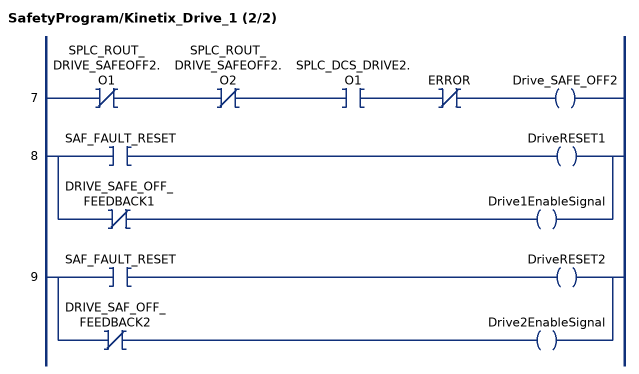
   7: XIO(SPLC_ROUT_DRIVE_SAFEOFF2.O1)XIO(SPLC_ROUT_DRIVE_SAFEOFF2.O2)XIC(SPLC_DCS_DRIVE2.O1)XIO(ERROR)OTE(Drive_SAFE_OFF2);
   8: [XIC(SAF_FAULT_RESET) OTE(DriveRESET1) ,XIO(DRIVE_SAFE_OFF_FEEDBACK1) OTE(Drive1EnableSignal) ];
   9: [XIC(SAF_FAULT_RESET) OTE(DriveRESET2) ,XIO(DRIVE_SAF_OFF_FEEDBACK2) OTE(Drive2EnableSignal) ];
END_ROUTINE

ROUTINE MainRoutine   (* ladder *)
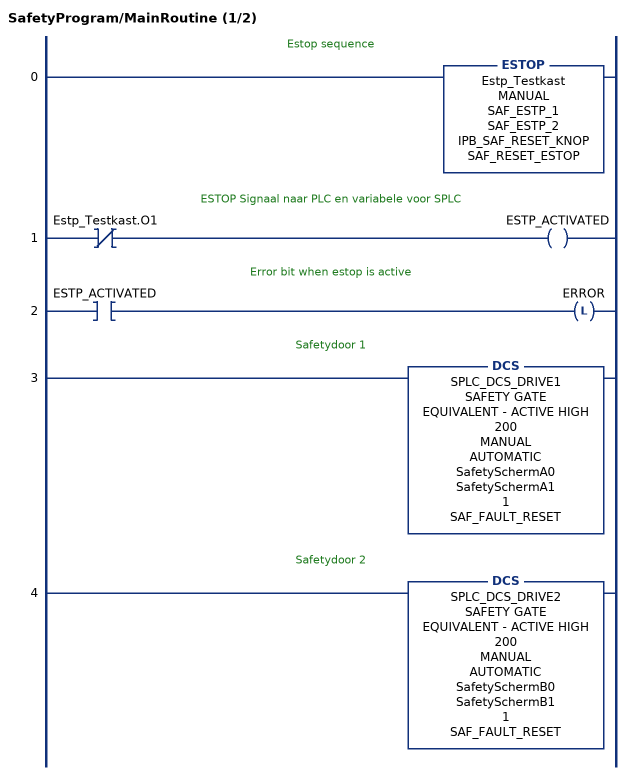
   // Estop sequence
   0: ESTOP(Estp_Testkast,MANUAL,SAF_ESTP_1,SAF_ESTP_2,IPB_SAF_RESET_KNOP,SAF_RESET_ESTOP);
   // ESTOP Signaal naar PLC en variabele voor SPLC
   1: XIO(Estp_Testkast.O1)OTE(ESTP_ACTIVATED);
   // Error bit when estop is active
   2: XIC(ESTP_ACTIVATED)OTL(ERROR);
   // Safetydoor 1
   3: DCS(SPLC_DCS_DRIVE1,SAFETY GATE,EQUIVALENT - ACTIVE HIGH,200,MANUAL,AUTOMATIC,SafetySchermA0,SafetySchermA1,1,SAF_FAULT_RESET);
   // Safetydoor 2
   4: DCS(SPLC_DCS_DRIVE2,SAFETY GATE,EQUIVALENT - ACTIVE HIGH,200,MANUAL,AUTOMATIC,SafetySchermB0,SafetySchermB1,1,SAF_FAULT_RESET);
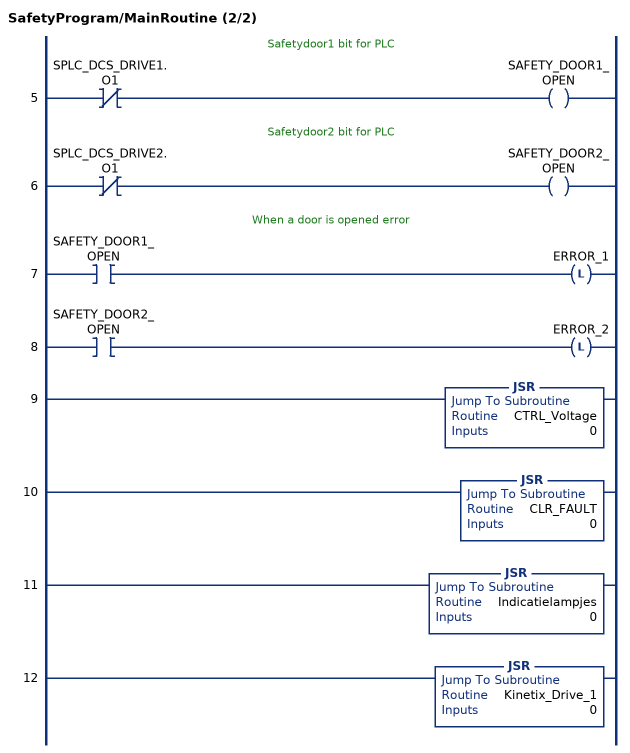
   // Safetydoor1 bit for PLC
   5: XIO(SPLC_DCS_DRIVE1.O1)OTE(SAFETY_DOOR1_OPEN);
   // Safetydoor2 bit for PLC
   6: XIO(SPLC_DCS_DRIVE2.O1)OTE(SAFETY_DOOR2_OPEN);
   // When a door is opened error
   7: XIC(SAFETY_DOOR1_OPEN)OTL(ERROR_1);
   8: XIC(SAFETY_DOOR2_OPEN)OTL(ERROR_2);
   9: JSR(CTRL_Voltage,0);
   10: JSR(CLR_FAULT,0);
   11: JSR(Indicatielampjes,0);
   12: JSR(Kinetix_Drive_1,0);
END_ROUTINE
END_PROGRAM
